{attribute 'qualified_only'}
{attribute 'strict'}
TYPE OvenSlider :
(
	retract := 0,
	extend,
	switchoff
);
END_TYPE

(* stored: Version 1.1.0.1, ProductVersion 3.1.4022.12
   DUT OvenSlider: Id {05984064-3f7b-410f-ad88-771c51fbfa5a} *)
